// Mitsubishi GX Works2 project: LRI_desafio_27.09   PLC: Q03UDV

PROGRAM MAIN
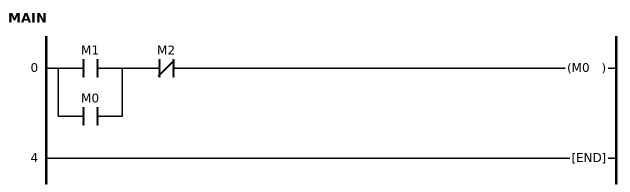
0     LD      M1
      OR      M0
      ANI     M2
      OUT     M0
4     END
END_PROGRAM
